(* CoDeSys 2.3 export: test3.exp *)
(* Libraries: ANALYZATION.LIB 5.10.99 09:05:06, IECSFC.LIB 13.4.06 15:51:28, STANDARD.LIB 4.10.05 11:14:46 *)

(* PLC configuration (modules and I/O channels)
PLC110_30 [Root] node -1, in %IB0 out %QB0 {param 1 = PLC110-30_v2; param 2 = 1; param 3 = 1000}
  Fast discrete inputs [I_SIMPLE_INPUT] node 0, in %IB0 out %QB0 {param 1 = Fast discrete inputs; param 2 = 10000}
    gEncoderA AT %IX0.0 [BitInput] Discrete input 1 {param 1 = Enter name}
    gEncoderB AT %IX0.1 [BitInput] Discrete input 2 {param 1 = Enter name}
  Discrete inputs - 16 [ID130] node 1, in %IB1 out %QB1 {param 1 = Discrete inputs; param 2 = 10; param 3 = 16}
    AT %IB1.0 [ByteInput] 8 discrete inputs {param 1 = Enter name}
    AT %IB1.1 [ByteInput] 8 discrete inputs {param 1 = Enter name}
  Fast discrete outputs [OWEN_ID570] node 2, in %IB2 out %QB2 {param 1 = Fast discrete outputs; param 2 = FALSE; param 3 = FALSE; param 4 = FALSE; param 5 = FALSE}
    gDO_1 AT %QX2.0 [BitOutput] Fast discrete output 1 {param 1 = Enter name}
    gDO_2 AT %QX2.1 [BitOutput] Fast discrete output 2 {param 1 = Enter name}
    gDO_3 AT %QX2.2 [BitOutput] Fast discrete output 3 {param 1 = Enter name}
    gDO_4 AT %QX2.3 [BitOutput] Fast discrete output 4 {param 1 = Enter name}
  Discrete outputs - 8 [ID131] node 3, in %IB3 out %QB3 {param 1 = Discrete outputs; param 2 = 0; param 3 = No; param 4 = 10}
    AT %QB3.0 [ByteOutput] 8 discrete outputs {param 1 = Enter name}
  Special input [ID103] node 4, in %IB4 out %QB4 {param 1 = Special input}
    AT %IX4.0 [BitInput] Special input {param 1 = Enter name}
  Special output [ID104] node 5, in %IB5 out %QB5 {param 1 = Special output}
    gBeeper AT %QX5.0 [BitOutput] Special output {param 1 = Enter name}
  ModBus (Master) [MODBUS_MASTER_ID450] node 6, in %IB6 out %QB6 {param 1 = ModBus (Master); param 2 = No}
    gModbus_Master_Channel AT %QD6.0 [DWordOutput] Last address {param 1 = Enter name}
    gModbus_Master_LastError AT %QW6.1 [WordOutput] Last error {param 1 = Enter name}
    RS-485-1 [COM1_USART] node 0, in %IB6.0 out %QB6.0 {param 1 = RS-485-1; param 2 = 9600; param 3 = NO PARITY CHECK; param 4 = 8 bits; param 5 = One stop bit; param 6 = RS485; param 7 = RTU; param 8 = 200; param 9 = No}
    Universal Modbus device [ID2000] node 1, in %IB6.1 out %QB6.1 {param 1 = ESP8266; param 2 = 10:0:0:223; param 3 = 150; param 4 = 502; param 5 = Serial; param 6 = 1; param 7 = By poll time; param 8 = 100; param 9 = No; param 10 = 0; param 11 = Trace_mode}
      AT %QB6.1.0 [ComChannel] Command (0xff - Start) {param 1 = Enter name}
      Register output module [ID2004] node 0, in %IB6.1.0 out %QB6.1.0 {param 1 = Register; param 2 = 0; param 3 = Write multiple registers(0x10); param 8 = No}
        mb_out_DefaultTarget AT %QW6.1.0.0 [WordOutput] {param 1 = Enter name}
      Register output module [ID2004] node 1, in %IB6.1.1 out %QB6.1.1 {param 1 = Register; param 2 = 1; param 3 = Write multiple registers(0x10); param 8 = No}
        mb_out_CurrentAngle AT %QW6.1.1.0 [WordOutput] {param 1 = Enter name}
      Register output module [ID2004] node 2, in %IB6.1.2 out %QB6.1.2 {param 1 = Register; param 2 = 2; param 3 = Write multiple registers(0x10); param 8 = No}
        mb_out_TargetAngle AT %QW6.1.2.0 [WordOutput] {param 1 = Enter name}
      Register output module [ID2004] node 3, in %IB6.1.3 out %QB6.1.3 {param 1 = Register; param 2 = 3; param 3 = Write multiple registers(0x10); param 8 = No}
        mb_out_Cycle AT %QW6.1.3.0 [WordOutput] {param 1 = Enter name}
      Register output module [ID2004] node 4, in %IB6.1.4 out %QB6.1.4 {param 1 = Register; param 2 = 4; param 3 = Write multiple registers(0x10); param 8 = No}
        mb_out_Done AT %QW6.1.4.0 [WordOutput] {param 1 = Enter name}
      Register output module [ID2004] node 5, in %IB6.1.5 out %QB6.1.5 {param 1 = Register; param 2 = 5; param 3 = Write multiple registers(0x10); param 8 = No}
        mb_out_Mode AT %QW6.1.5.0 [WordOutput] {param 1 = Enter name}
      Register output module [ID2004] node 6, in %IB6.1.6 out %QB6.1.6 {param 1 = Register; param 2 = 6; param 3 = Write multiple registers(0x10); param 8 = No}
        mb_out_Pedals AT %QW6.1.6.0 [WordOutput] {param 1 = Enter name}
      Register input module [ID2003] node 7, in %IB6.1.7 out %QB6.1.7 {param 1 = Register input module; param 2 = 9; param 3 = Read holding Registers  (0x03); param 8 = No}
        mb_in_Command AT %QW6.1.7.0 [WordOutput] {param 1 = Enter name}
      Register input module [ID2003] node 8, in %IB6.1.8 out %QB6.1.8 {param 1 = Register input module; param 2 = 10; param 3 = Read holding Registers  (0x03); param 8 = No}
        mb_in_WebTarget AT %QW6.1.8.0 [WordOutput] {param 1 = Enter name}
*)

(* Global variable list: Global_Variables *)
VAR_GLOBAL RETAIN
    gTargetAngle : REAL := 45.0;
    gDefaultTarget : REAL := 45.0;
    gCurrentAngle : REAL := 0.0;
    gCycle : INT := 1;
    gEncoderCount : DINT := 0;
    gCalibCountsPerRev : DINT := 360;

    gCalibStatus : INT := 0;
    gCalibRevsDone : INT := 0;
    gCalibRevsTarget : INT := 3;
    gCalibMeasured : REAL := 0.0;

    (* Modbus / system variables and Modbus-mapped registers are defined by PLC_CONFIGURATION;
       do not redeclare `gModbus_Master_*`, `mb_out_*` or `mb_in_*` here to avoid duplicates. *)
    (* gDI and gDO variables are also typically defined in PLC_CONFIGURATION *)
END_VAR

(* Data type *)
TYPE COMSETTINGS_FALLBACK : STRUCT
    Port : INT; (* PORTS in library; INT used locally to avoid enum conflicts *)
    dwBaudRate : DWORD;
    byStopBits : BYTE;
    byParity : BYTE;
    dwTimeout : DWORD;
    dwBufferSize : DWORD;
    dwScan : DWORD;
END_STRUCT
END_TYPE

(* POU PLC_PRG, ST *)
PROGRAM PLC_PRG
VAR
    (* Control Inputs *)
    prev_d5 : BOOL := TRUE;  (* Edge detection for Manual/Auto switch *)
    enableStart : BOOL;      (* Manual Mode (TRUE) / Auto Mode (FALSE) *)
    
    (* Pedals *)
    btnD7 : BOOL;            (* Forward *)
    btnD8 : BOOL;            (* Backward *)
    both : BOOL;             (* Both pressed *)
    
    prev_d7 : BOOL := FALSE;
    prev_d8 : BOOL := FALSE;
    prev_both : BOOL := FALSE;

    (* Encoder *)
    encAEdge : R_TRIG;
    encBEdge : R_TRIG;

    (* Process State *)
    done : BOOL := FALSE;    (* Target reached flag *)
    
    (* Timers & Triggers *)
    targetPulseTrigger : BOOL := FALSE;
    tpTarget : TP;           (* Done Pulse *)
    
    beepTargetTrigger : BOOL := FALSE;
    tpBeepTarget : TP;       (* Done Beep *)

    (* Error Beep Logic *)
    errorBeepTrigger : BOOL := FALSE;
    tErrTotal : TON;
    tErrDelay1 : TON;
    tErrDelay2 : TON;
    tErrDelay3 : TON;
    rTrigErr1 : R_TRIG;
    rTrigErr2 : R_TRIG;
    rTrigErr3 : R_TRIG;
    tpErr : TP;

    (* Modbus / Web control *)
    prev_mb_in_command : WORD := 0;
    prev_mb_in_WebTarget : WORD := 0;
    init_done : BOOL := FALSE;
    
    (* Helper for Modbus Output Mapping *)
    (* Ensure global vars are assigned to outputs if mapped there *)
END_VAR
(* 1. Input Mapping *)
enableStart := gDI_5;
btnD7 := gDI_7;
btnD8 := gDI_8;
both := btnD7 AND btnD8;

(* 2. Encoder Processing *)
encAEdge(CLK := gEncoderA);
(* encBEdge(CLK := gEncoderB); Not typically needed for quadrature decoding if using A edge + B level *)

IF encAEdge.Q THEN
    IF gEncoderB THEN
        (* Direction depends on wiring, assuming B leads or lags *)
        (* Adjust +/- based on empirical test if counting wrong direction *)
        gEncoderCount := gEncoderCount + 1;
    ELSE
        gEncoderCount := gEncoderCount - 1;
    END_IF;
END_IF;

(* 3. Angle Calculation *)
IF gCalibCountsPerRev = 0 THEN gCalibCountsPerRev := 360; END_IF;
(* Negative sign to align physical direction with logical angle increases *)
gCurrentAngle := -1.0 * (DINT_TO_REAL(gEncoderCount) * 360.0 / DINT_TO_REAL(gCalibCountsPerRev));

(* 4. Mode Switching & Calibration *)
(* When switching from Manual (1) to Auto (0), resetting zero position *)
IF (prev_d5 AND NOT enableStart) THEN
    gEncoderCount := 0;
    gCurrentAngle := 0.0;
    gCycle := 1;
    gTargetAngle := gDefaultTarget;
    done := FALSE;
END_IF;
prev_d5 := enableStart;

(* 5. Modbus / Web Commands Processing *)

(* 5.1 Web Target Update *)
(* If WebTarget changes, update logical target *)
IF mb_in_WebTarget <> prev_mb_in_WebTarget THEN
    IF init_done THEN (* Avoid overwriting on startup if ESP is 0 *)
         gDefaultTarget := WORD_TO_REAL(mb_in_WebTarget) / 10.0;
         gTargetAngle := gDefaultTarget; 
         gCycle := 1;
         done := FALSE;
    ELSE
         (* Sync local previous value to current input on first scan to establish baseline *)
         (* If ESP sends 0 on startup, we ignore it as a 'change' for the logic, 
            presuming RETAIN gDefaultTarget is correct. *)
         NULL; 
    END_IF;
END_IF;
prev_mb_in_WebTarget := mb_in_WebTarget;
init_done := TRUE;

(* 5.2 Command Register *)
IF mb_in_Command <> 0 AND mb_in_Command <> prev_mb_in_command THEN
    CASE WORD_TO_INT(mb_in_Command) OF
        1: (* START *)
            IF NOT enableStart THEN 
                done := FALSE; 
                gCycle := 1; 
                gTargetAngle := gDefaultTarget;
            END_IF;
        2: (* STOP *)
            (* Just stops motors by logic below, setting done=TRUE effectively stops Auto moves *)
             (* But STOP usually means emergency stop. In Auto, we can set Done=TRUE to stop. *)
             done := TRUE;
        3: (* ZERO / CALIBRATE *)
            gEncoderCount := 0;
            gCurrentAngle := 0.0;
    END_CASE;
END_IF;
prev_mb_in_command := mb_in_Command;

(* 6. Cycle Logic (Auto Mode) *)
IF NOT enableStart AND NOT done THEN
    IF gCycle = 1 THEN
        gTargetAngle := gDefaultTarget;
    ELSIF gCycle = 2 THEN
        gTargetAngle := 0.0;
    END_IF;
END_IF;

(* 7. Output to Modbus (Mapping to Output Registers) *)
mb_out_DefaultTarget := REAL_TO_WORD(gDefaultTarget * 10.0);
mb_out_CurrentAngle  := REAL_TO_WORD(ABS(gCurrentAngle * 10.0));
mb_out_TargetAngle   := REAL_TO_WORD(gTargetAngle * 10.0);
mb_out_Cycle         := INT_TO_WORD(gCycle);

IF done THEN mb_out_Done := 1; ELSE mb_out_Done := 0; END_IF;
IF enableStart THEN mb_out_Mode := 1; ELSE mb_out_Mode := 0; END_IF;

mb_out_Pedals := 0;
IF btnD7 THEN mb_out_Pedals := mb_out_Pedals + 1; END_IF;
IF btnD8 THEN mb_out_Pedals := mb_out_Pedals + 2; END_IF;

(* 8. Motor Control Logic *)
(* gDO_10 = Forward, gDO_11 = Backward *)

IF enableStart THEN  (* MANUAL MODE *)
    IF both THEN
        gDO_10 := FALSE;
        gDO_11 := FALSE;
    ELSE
        gDO_10 := btnD7;
        gDO_11 := btnD8;
    END_IF;
ELSE  (* AUTO MODE *)
    (* Move Forward if: Pedal Fwd, Not Back, Angle < Target, Not Done *)
    gDO_10 := btnD7 AND NOT btnD8 AND NOT both AND (gCurrentAngle < gTargetAngle) AND NOT done;
    
    (* Move Backward if: Pedal Back, Not Fwd, Angle > 0, Not Done, Not Both *)
    gDO_11 := btnD8 AND NOT btnD7 AND NOT both AND (gCurrentAngle > 0.0) AND NOT done;
END_IF;

(* 9. Target Reached Check *)
IF NOT enableStart AND NOT done THEN
    IF ABS(gCurrentAngle - gTargetAngle) < 0.5 THEN
        done := TRUE;
        targetPulseTrigger := TRUE;
        beepTargetTrigger := TRUE;
        (* Switch Cycle for next move *)
        IF gCycle = 1 THEN gCycle := 2; ELSE gCycle := 1; END_IF;
    END_IF;
END_IF;

(* Re-enable movement if drift occurs? Or wait for next command? 
   TZ says: "If after this deviation exceeds 1 deg, done resets" *)
IF ABS(gCurrentAngle - gTargetAngle) > 1.0 THEN
    done := FALSE;
END_IF;

(* 10. Indication & Beeper *)

(* Target Pulse (DO_12) *)
tpTarget(IN := targetPulseTrigger, PT := T#500MS);
gDO_12 := tpTarget.Q;
IF tpTarget.Q THEN targetPulseTrigger := FALSE; END_IF;

(* Target Beep *)
tpBeepTarget(IN := beepTargetTrigger, PT := T#500MS);
IF tpBeepTarget.Q THEN beepTargetTrigger := FALSE; END_IF;

(* Error Conditions *)
IF NOT enableStart THEN
    (* Error: Forward pedal when already at/past target *)
    IF (btnD7 AND NOT prev_d7) AND (gCurrentAngle >= gDefaultTarget) AND (gCycle = 1) THEN
        errorBeepTrigger := TRUE;
    END_IF;
    (* Error: Back pedal when already at 0 *)
    IF (btnD8 AND NOT prev_d8) AND (gCurrentAngle <= 0.0) AND (gCycle = 2) THEN
        errorBeepTrigger := TRUE;
    END_IF;
    (* Error: Both pedals *)
    IF both AND NOT prev_both THEN
        errorBeepTrigger := TRUE;
    END_IF;
END_IF;

(* Error Beep Sequence (3 short beeps) *)
tErrTotal(IN := errorBeepTrigger, PT := T#1400MS);
tErrDelay1(IN := errorBeepTrigger, PT := T#0MS);
tErrDelay2(IN := errorBeepTrigger, PT := T#400MS);
tErrDelay3(IN := errorBeepTrigger, PT := T#800MS);

rTrigErr1(CLK := tErrDelay1.Q);
rTrigErr2(CLK := tErrDelay2.Q);
rTrigErr3(CLK := tErrDelay3.Q);

tpErr(IN := (rTrigErr1.Q OR rTrigErr2.Q OR rTrigErr3.Q), PT := T#200MS);

gBeeper := tpBeepTarget.Q OR tpErr.Q;

IF tErrTotal.Q THEN errorBeepTrigger := FALSE; END_IF;

(* Update Previous States *)
prev_d7 := btnD7;
prev_d8 := btnD8;
prev_both := both;
END_PROGRAM
